FUNCTION_BLOCK Integrator
VAR_INPUT
	ssMethodType: SINT;
	fSignal: LREAL;
END_VAR
VAR_OUTPUT
	fSignalIntegrated: LREAL;
END_VAR
VAR
	c_DiscreteTimeIntegrator_DS: LREAL;
END_VAR



CASE ssMethodType OF
    SS_INITIALIZE: 
        (* SystemInitialize for Atomic SubSystem: '<Root>/Integrator' *)
        (* InitializeConditions for DiscreteIntegrator: '<S1>/Discrete-Time Integrator' *)
        c_DiscreteTimeIntegrator_DS := 0.0;
        (* End of SystemInitialize for SubSystem: '<Root>/Integrator' *)
    SS_STEP: 
        (* Outputs for Atomic SubSystem: '<Root>/Integrator' *)
        (* Outport: '<Root>/fSignalIntegrated' incorporates:
         *  DiscreteIntegrator: '<S1>/Discrete-Time Integrator' *)
        fSignalIntegrated := c_DiscreteTimeIntegrator_DS;
        (* Update for DiscreteIntegrator: '<S1>/Discrete-Time Integrator' *)
        c_DiscreteTimeIntegrator_DS := (0.001 * fSignal) + c_DiscreteTimeIntegrator_DS;
        (* End of Outputs for SubSystem: '<Root>/Integrator' *)
END_CASE;

END_FUNCTION_BLOCK

(* stored: Version 1.1.0.1
   POU Integrator: Id {1200ebea-d33a-4080-b39f-2edfc1602a4c}, SpecialFunc None *)
